FUNCTION FC_Comms2

VAR_INPUT
	ix_Safety : BOOL := FALSE;	
	b_startBeweging : BOOL;
	
END_VAR
VAR
END_VAR
VAR_OUTPUT
	qx_E_Stop : BOOL;
	qx_StartBeweging : BOOL;
END_VAR



(*DB10_Alias.qx_kukaCommEstop:=FC_Comms2.qx_E_Stop;
DB10_Alias.qx_kukaComm2:=FC_Comms2.qx_StartBeweging;*)

END_FUNCTION

(* stored: Version 1.1.0.1, ProductVersion 3.1.4024.12
   POU FC_Comms2: Id {1e780b85-bf07-42d1-94f1-a6941c80cb9c}, SpecialFunc None *)
